// This function has been automatically generated from the project information.
{attribute 'signature_flag' := '1073741824'}
{attribute 'TcGenerated'}
{attribute 'no-analysis'}
FUNCTION F_GetTitle : WSTRING
VAR_INPUT
	
END_VAR

F_GetTitle := "Base Library";

END_FUNCTION

(* stored: Version 1.1.0.1
   POU F_GetTitle: Id {fe7ec784-4b77-4a99-941d-edd02cb0b34a}, SpecialFunc None *)
